// TIA Portal V18 export
// export: Created 2026-03-12T16:04:35.8661033Z, ExportSetting WithDefaults, DisplayName Totally Integrated Automation Portal, DisplayVersion V18 Update 5, DisplayName TIA Portal Openness, DisplayVersion V18 Update 5, DisplayName TIA Portal Version Control Interface, DisplayVersion V18, DisplayName SINAMICS Startdrive Advanced, DisplayVersion V18, DisplayName SINAMICS Startdrive G130, G150, S120, S150, SINAMICS MV, S210, DisplayVersion V18, DisplayName SINAMICS Startdrive G110M, G120, G120C, G120D, G120P, G115D, DisplayVersion V18, DisplayName STEP 7 Professional, DisplayVersion V18 Update 5, DisplayName STEP 7 Safety, DisplayVersion V18, DisplayName WinCC Professional, DisplayVersion V18 Update 5
FUNCTION_BLOCK "FB_MOVE_DRIVE_DANFOSS"   // FB31, SCL
{ S7_Optimized_Access := 'TRUE' }
VERSION : 0.1
// stored: AutoNumber true, IsIECCheckEnabled false, IsRetainMemResEnabled false, MemoryReserve 100, SetENOAutomatically false, UDAEnableTagReadback false
   VAR_INPUT
      IN_1 : Array[1..8] of UInt;
      IN_2 : Array[1..8] of UInt;
      IN_3 : Array[1..8] of UInt;
      IN_4 : Array[1..8] of UInt;
      IN_5 : Array[1..8] of UInt;
      IN_6 : Array[1..8] of UInt;
   END_VAR
   VAR_IN_OUT
      OUT_1 : "MotorDados";
      OUT_2 : "MotorDados";
      OUT_3 : "MotorDados";
      OUT_4 : "MotorDados";
      OUT_5 : "MotorDados";
      OUT_6 : "MotorDados";
   END_VAR
BEGIN
   // ===============================
   // DISPOSITIVO 1
   // ===============================
   #OUT_1.POTENCIA := UINT_TO_INT(#IN_1[1]);
   #OUT_1.REF_VELOCIDADE := (UINT_TO_REAL(#IN_1[2]))/10;
   #OUT_1.CORRENTE := (UINT_TO_REAL (#IN_1[3])/10);

   // ===============================
   // DISPOSITIVO 2
   // ===============================
   #OUT_2.POTENCIA := UINT_TO_INT(#IN_2[1]);
   #OUT_2.REF_VELOCIDADE := (UINT_TO_REAL(#IN_2[2]))/10;
   #OUT_2.CORRENTE := (UINT_TO_REAL (#IN_2[3])/10);

   // ===============================
   // DISPOSITIVO 3
   // ===============================
   #OUT_3.POTENCIA := UINT_TO_INT(#IN_3[1]);
   #OUT_3.VELOCIDADE := (UINT_TO_INT(#IN_3[2])/10);
   #OUT_3.CORRENTE := (UINT_TO_REAL (#IN_3[3])/10);

   // ===============================
   // DISPOSITIVO 4
   // ===============================
   #OUT_4.POTENCIA := UINT_TO_INT(#IN_4[1]);
   #OUT_4.VELOCIDADE := (UINT_TO_INT(#IN_4[2])/10);
   #OUT_4.CORRENTE := (UINT_TO_REAL (#IN_4[3])/10);

   // ===============================
   // DISPOSITIVO 5
   // ===============================
   #OUT_5.POTENCIA := UINT_TO_INT(#IN_5[1]);
   #OUT_5.VELOCIDADE := UINT_TO_INT(#IN_5[2])/10;
   #OUT_5.CORRENTE := (UINT_TO_REAL (#IN_5[3])/10);

   // ===============================
   // DISPOSITIVO 6
   // ===============================
   #OUT_6.POTENCIA := UINT_TO_INT(#IN_6[1]);
   #OUT_6.VELOCIDADE := (UINT_TO_INT(#IN_6[2])/10);
   #OUT_6.CORRENTE := (UINT_TO_REAL (#IN_6[3])/10);
END_FUNCTION_BLOCK
